(* CODESYS project task9.project
   Title: Adsız
   Version: 0.0.0.0
   Author: USER

Project tree, tasks and I/O mapping:
  MyController : TM238LFDC24DT, Schneider Electric, order no. TM238LFDC24DT, version 4.0.1.28
      settings: OpcUa Enable = False
    application Application
      task MAST (cyclic, interval 20 ms, priority 15, watchdog 100 ms x 1) calls POU
      global variables GVL
      program POU [LD]
    Embedded Functions
      IO : IO, Schneider Electric, version 4.0.1.28
          input  sensor1 : BOOL  // IW0.I0
          input  button1 : BOOL  // IW0.I1
          input  button2 : BOOL  // IW0.I2
          input  sensor2 : BOOL  // IW0.I3
          output motor : BOOL  // QW0.Q2
          output servomotor : BOOL  // QW0.Q3
          unmapped channels: IW0, QW0
      HSC : HSC, Schneider Electric, version 4.0.1.28
      PTO_PWM : PTO_PWM, Schneider Electric, version 4.0.1.28
    Serial Line 1
      Modbus_Manager : Modbus Manager, Schneider Electric, version 4.0.0.2
    Serial Line 2
      SoMachine_Network_Manager : SoMachine-Network Manager, Schneider Electric, version 4.0.0.2
    CAN
*)

// MyController/Application/GVL
VAR_GLOBAL
END_VAR

// MyController/Application/POU
PROGRAM POU
VAR
	motor: BOOL;
	button1: BOOL;
	sensor1: BOOL;
	sensor2: BOOL;
	servomotor: BOOL;
	button2: BOOL;
	cv1: WORD;
	et1: TIME;
	ton_1: TON;
	ctu_1: CTU;
END_VAR

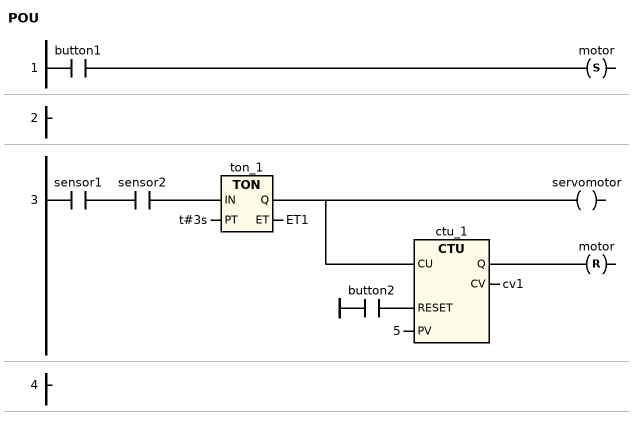
// NETWORK 1
motor S= button1;

// NETWORK 2

// NETWORK 3
ton_1(IN := sensor1 AND sensor2, PT := t#3s, ET => ET1); // TON
servomotor := ton_1.Q;
ctu_1(CU := ton_1.Q, RESET := button2, PV := 5, CV => cv1); // CTU
motor R= ctu_1.Q;

// NETWORK 4

END_PROGRAM
